// TIA Portal V16 program export: 1 tag tables, 0 data types, 2 data blocks, 4 code blocks (in call order from the OBs), 2 instance data blocks

VAR_GLOBAL   // PLC tag table "Default tag table"
END_VAR

DATA_BLOCK "DI"   // DB1
{ S7_Optimized_Access := 'TRUE' }
VERSION : 0.1
// stored: AutoNumber true, IsOnlyStoredInLoadMemory false, IsRetainMemResEnabled false, IsWriteProtectedInAS false, MemoryReserve 100
   VAR
      xCzujnikKrancowyNoza : Bool;
      xResetLicznika : Bool;
   END_VAR
BEGIN
END_DATA_BLOCK

DATA_BLOCK "DO"   // DB2
{ S7_Optimized_Access := 'TRUE' }
VERSION : 0.1
// stored: AutoNumber true, IsOnlyStoredInLoadMemory false, IsRetainMemResEnabled false, IsWriteProtectedInAS false, MemoryReserve 100
   VAR
      xLampkaCzerwona : Bool;
      xLampkaZielona : Bool;
   END_VAR
BEGIN
END_DATA_BLOCK

ORGANIZATION_BLOCK "Main"   // OB1, LAD, ProgramCycle
TITLE = "Main Program Sweep (Cycle)"
{ S7_Optimized_Access := 'TRUE' }
VERSION : 0.1
// stored: AutoNumber true, IsIECCheckEnabled false, SetENOAutomatically false
   VAR_INPUT
      Initial_Call : Bool;   // Initial call of this OB
      Remanence : Bool;   // =True, if remanent data are available
   END_VAR
BEGIN

REGION Network 1
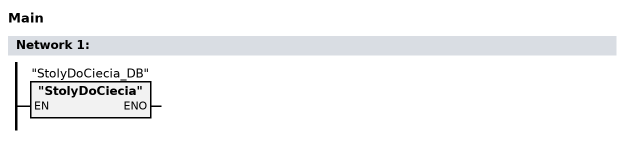
   RUNG wire#powerrail
      "StolyDoCiecia_DB"()
   END_RUNG
   // the same network as SCL:
   "StolyDoCiecia_DB"();   // "StolyDoCiecia"
END_REGION
END_ORGANIZATION_BLOCK

FUNCTION_BLOCK "StolyDoCiecia"
{ S7_Optimized_Access := 'TRUE' }
VERSION : 0.1

BEGIN
	//wywołanie bloku funkcyjnego dla 1 stołu
	"StanowiskoCiecia_1_DB"(xSygnalWyzwalajacy:="DI".xCzujnikKrancowyNoza,
	                        xResetLicznika:="DI".xResetLicznika,
	                        xZlecenieWToku=>"DO".xLampkaZielona,
	                        xZlecenieZakonczone=>"DO".xLampkaCzerwona);
	
	
END_FUNCTION_BLOCK

FUNCTION_BLOCK "StanowiskoCiecia"
{ S7_Optimized_Access := 'TRUE' }
VERSION : 0.1
   VAR_INPUT 
      iLiczbaCiecZadana : Int;
      xSygnalWyzwalajacy : Bool;
      xResetLicznika : Bool;
   END_VAR

   VAR_OUTPUT 
      xZlecenieWToku : Bool;
      xZlecenieZakonczone : Bool;
   END_VAR

   VAR_IN_OUT 
      iLicznikCiec : Int;
   END_VAR

   VAR 
      xBitPamieci : Bool;
   END_VAR


BEGIN
	// Wykrycie zbocza opadającego sygnalu noża oraz inkrementacja licznika
	#iLicznikCiec := #iLicznikCiec + BOOL_TO_INT(NOT #xSygnalWyzwalajacy AND #xBitPamieci);
	
	// Reset licznika
	#iLicznikCiec := #iLicznikCiec * BOOL_TO_INT(NOT #xResetLicznika);
	
	// Wizualizacja statusu zlecenia
	#xZlecenieWToku := #iLicznikCiec < #iLiczbaCiecZadana;
	#xZlecenieZakonczone := NOT #xZlecenieWToku;
	
	#xBitPamieci := #xSygnalWyzwalajacy;
END_FUNCTION_BLOCK

FUNCTION_BLOCK "Testowy"
{ S7_Optimized_Access := 'TRUE' }
VERSION : 0.1

BEGIN
END_FUNCTION_BLOCK

DATA_BLOCK "StanowiskoCiecia_1_DB"   // DB3
VERSION : 0.1
// stored: AutoNumber true, InstanceOfName StanowiskoCiecia, InstanceOfType FB
"StanowiskoCiecia"
BEGIN
END_DATA_BLOCK

DATA_BLOCK "StolyDoCiecia_DB"   // DB4
VERSION : 0.1
// stored: AutoNumber true, InstanceOfName StolyDoCiecia, InstanceOfType FB
"StolyDoCiecia"
BEGIN
END_DATA_BLOCK
